// TIA Portal V19 export
TYPE "udt_DeviceSafetyInterface"
// stored: Access Published, IsFailsafeCompliant true
   STRUCT
      SafeStop : Bool;
      PowerEnable : Bool;
      DevicesInSafeState : Bool;
   END_STRUCT;
END_TYPE
